PROGRAM MAIN
VAR
	a:INT;
	b:INT;
	c:INT;
	
	enable: BOOL;
END_VAR


IF enable THEN
	c:=a+b;
ELSE
	c:=0;
END_IF

END_PROGRAM

(* stored: Version 1.1.0.1, ProductVersion 3.1.4024.9
   POU MAIN: Id {6dd4f5eb-60fa-4e7b-ab23-f07ecac8c1c3}, SpecialFunc None *)
